FUNCTION_BLOCK TTestEvent_UsesEventArgs EXTENDS TEventBase 
VAR
    Handler : ITestEventHandler_UsesEventArgs;
END_VAR

METHOD PRIVATE CallHandler
VAR_INPUT
    HandlerBase : IEventHandlerBase;
    EventArgs   : IStreamReader;
END_VAR
IF __QUERYINTERFACE(HandlerBase,Handler) THEN
    Handler.OnThisEvent(EventArgs);
//ELSE
//    tcl_BaseClasses.F_LogError('Event Handling',F_FormatStringEx1('Error raising %s - invalid handler',EventName));
END_IF
END_METHOD

METHOD IsHandlerSupported : BOOL
VAR_INPUT
    HandlerBase : IEventHandlerBase;
END_VAR
IF __QUERYINTERFACE(HandlerBase,Handler) THEN
    IsHandlerSupported := TRUE;
END_IF
END_METHOD

END_FUNCTION_BLOCK

(* stored: Version 1.1.0.1, ProductVersion 3.1.4024.4
   POU TTestEvent_UsesEventArgs: Id {306ef5b7-3bc3-4016-b308-fa1f9ccb4bd0}, SpecialFunc None
   Method CallHandler: Id {cc3d4fe9-0b2e-4d79-9506-a46fc5059d65}
   Method IsHandlerSupported: Id {21ce5b3f-d70d-40ee-8278-ec060633ed10} *)
